(* IEC 61131-3 sources: Word/plc-course/13-sequential-control/labs/starter, 3 files *)

(* ---- 13-1-pedestrian-crossing.st ---- *)
(* Lab 13-1: Pedestrian crossing as a CASE state machine.
   Module 13 (Sequential control). STARTER - the declarations are done for you;
   write the logic where it says TODO, then run:
     python3 tools/plctest.py 13-sequential-control/labs/starter/13-1-pedestrian-crossing.st

   The enumeration, the state variables and the step timer are suggestions:
   the test only looks at the I/O and the settings, so you may organise the
   internals differently. *)

TYPE
  E_Crossing : (Startup, RedAmber, Green, Amber, AllRed, Walk, PedClear);
END_TYPE

PROGRAM PedCrossing
  VAR (* I/O *)
    PedPB    AT %IX0.0 : BOOL;  (* pedestrian request push-button, NO *)
    CarRed   AT %QX0.0 : BOOL;  (* vehicle signal, red *)
    CarAmber AT %QX0.1 : BOOL;  (* vehicle signal, amber *)
    CarGreen AT %QX0.2 : BOOL;  (* vehicle signal, green *)
    PedRed   AT %QX0.3 : BOOL;  (* pedestrian signal, red figure: do not cross *)
    PedGreen AT %QX0.4 : BOOL;  (* pedestrian signal, green figure: cross *)
    WaitLamp AT %QX0.5 : BOOL;  (* WAIT lamp on the push-button box *)
  END_VAR
  VAR (* settings *)
    StartupTime  : TIME := T#3s;   (* all red after power-up *)
    RedAmberTime : TIME := T#2s;   (* red + amber before green *)
    MinGreen     : TIME := T#10s;  (* minimum vehicle green *)
    AmberTime    : TIME := T#3s;   (* amber after green *)
    AllRedTime   : TIME := T#2s;   (* all red before the walk phase *)
    WalkTime     : TIME := T#6s;   (* steady green figure *)
    PedClearTime : TIME := T#4s;   (* flashing green figure *)
  END_VAR
  VAR (* internal - add your own helper variables here *)
    State      : E_Crossing := E_Crossing#Startup;
    PrevState  : E_Crossing := E_Crossing#Startup;
    FirstScan  : BOOL := TRUE;
    StepEntry  : BOOL;           (* TRUE on the first scan in a state *)
    StepTimer  : TON;            (* time spent in the current state *)
    Request    : BOOL;           (* latched pedestrian request *)
    FlashTimer : TON;            (* 500 ms flasher for the clearance phase *)
    FlashOn    : BOOL;
  END_VAR

  (* TODO: replace these placeholder lines with your logic.
     1. Step bookkeeping: StepEntry and StepTimer (reset on every change).
     2. CASE State OF ... with the transitions of each state.
     3. The request latch and the flasher.
     4. One assignment per output, derived from State. *)
  CarRed := TRUE;
  CarAmber := FALSE;
  CarGreen := FALSE;
  PedRed := TRUE;
  PedGreen := FALSE;
  WaitLamp := FALSE;
END_PROGRAM

CONFIGURATION Config0
  RESOURCE Res0 ON PLC
    TASK MainTask(INTERVAL := T#10ms, PRIORITY := 0);
    PROGRAM Inst0 WITH MainTask : PedCrossing;
  END_RESOURCE
END_CONFIGURATION

(* ---- 13-2-batch-tank.st ---- *)
(* Lab 13-2: Batch tank sequence with watchdogs, Hold/Resume and Abort.
   Module 13 (Sequential control). STARTER - the declarations are done for you;
   write the logic where it says TODO, then run:
     python3 tools/plctest.py 13-sequential-control/labs/starter/13-2-batch-tank.st

   The enumeration and the internal variables are suggestions: the test only
   looks at the I/O, TankTemp, the settings, FaultCode and BatchCount. *)

TYPE
  E_Batch : (Idle, Filling, Mixing, Heating, Draining, Complete, Held, Faulted);
END_TYPE

PROGRAM BatchTank
  VAR (* I/O *)
    StartPB      AT %IX0.0 : BOOL;  (* start a batch, NO *)
    HoldPB       AT %IX0.1 : BOOL;  (* hold the batch, NO *)
    ResumePB     AT %IX0.2 : BOOL;  (* resume a held batch, NO *)
    AbortPB      AT %IX0.3 : BOOL;  (* abort the batch, NO *)
    ResetPB      AT %IX0.4 : BOOL;  (* fault reset, NO *)
    LevelHighLS  AT %IX0.5 : BOOL;  (* high-level switch: TRUE when the tank is full *)
    LevelLowLS   AT %IX0.6 : BOOL;  (* low-level switch: TRUE while liquid covers it (and the heater) *)
    InletValve   AT %QX0.0 : BOOL;  (* fill valve *)
    Agitator     AT %QX0.1 : BOOL;  (* mixer motor *)
    Heater       AT %QX0.2 : BOOL;  (* immersion heater contactor *)
    OutletValve  AT %QX0.3 : BOOL;  (* drain valve *)
    RunLamp      AT %QX0.4 : BOOL;  (* batch running *)
    HeldLamp     AT %QX0.5 : BOOL;  (* batch held *)
    FaultLamp    AT %QX0.6 : BOOL;  (* sequence fault *)
    CompleteLamp AT %QX0.7 : BOOL;  (* batch complete *)
  END_VAR
  VAR (* process value, written by the analog-input layer (Module 14) *)
    TankTemp : REAL;                (* tank temperature, degC *)
  END_VAR
  VAR (* settings *)
    TempSP       : REAL := 60.0;    (* heat until TankTemp >= TempSP *)
    MixTime      : TIME := T#10s;   (* total mixing time *)
    FillTimeout  : TIME := T#30s;   (* watchdog: filling *)
    HeatTimeout  : TIME := T#60s;   (* watchdog: heating *)
    DrainTimeout : TIME := T#30s;   (* watchdog: draining *)
  END_VAR
  VAR (* status for the HMI *)
    FaultCode  : INT;               (* 0 none, 1 fill, 2 heat, 3 drain timeout *)
    BatchCount : INT;               (* completed batches *)
  END_VAR
  VAR (* internal - suggestions; add or change as you like *)
    State     : E_Batch := Idle;
    PrevState : E_Batch := Idle;
    HeldFrom  : E_Batch := Idle;  (* the step to resume *)
    FirstScan : BOOL := TRUE;
    StepEntry : BOOL;               (* TRUE on the first scan in a state *)
    StepTimer : TON;                (* time in the current state *)
    MixDone   : TIME;               (* mixing completed before a hold *)
    Running   : BOOL;               (* in one of the four process steps *)
    (* One instance per line: OpenPLC's compiler can crash on a list of
       FB instances in one declaration (see Appendix E). *)
    StartEdge : R_TRIG;
    HoldEdge : R_TRIG;
    ResumeEdge : R_TRIG;
    AbortEdge : R_TRIG;
    ResetEdge : R_TRIG;
    StartCmd, HoldCmd, ResumeCmd, AbortCmd, ResetCmd : BOOL;
  END_VAR

  (* TODO: replace these placeholder lines with your logic.
     1. Operator commands on the rising edge (R_TRIG).
     2. Step bookkeeping: StepEntry and StepTimer, reset on every change.
     3. Entry actions (BatchCount), before the transitions.
     4. Transitions: Abort first, then Hold, then CASE State OF ...
        with a watchdog in Filling, Heating and Draining.
     5. One assignment per output, derived from State, plus the heater and
        inlet interlocks. *)
  InletValve := FALSE;
  Agitator := FALSE;
  Heater := FALSE;
  OutletValve := FALSE;
  RunLamp := FALSE;
  HeldLamp := FALSE;
  FaultLamp := FALSE;
  CompleteLamp := FALSE;
END_PROGRAM

CONFIGURATION Config0
  RESOURCE Res0 ON PLC
    TASK MainTask(INTERVAL := T#10ms, PRIORITY := 0);
    PROGRAM Inst0 WITH MainTask : BatchTank;
  END_RESOURCE
END_CONFIGURATION

(* ---- 13-3-drill-sfc.st ---- *)
(* Lab 13-3: Drilling station in textual SFC, with action qualifiers.
   Module 13 (Sequential control). STARTER - the declarations are done for you;
   write the chart where it says TODO, then run:
     python3 tools/plctest.py 13-sequential-control/labs/starter/13-3-drill-sfc.st

   The program body is a Sequential Function Chart in the textual form of
   IEC 61131-3. Only the initial step is written so far. Add the steps,
   transitions and actions described in the lab, for example:

     STEP Clamp:
       ClampValve(S);
     END_STEP

     TRANSITION FROM Idle TO Clamp
       := StartPB AND PartPE AND DrillUpLS;
     END_TRANSITION

     ACTION CountHole:
       HoleCount := HoleCount + 1;
     END_ACTION

   Remember: a step name cannot be the same as a variable name, and two
   transitions leaving the same step must never be TRUE together. *)

PROGRAM DrillCycle
  VAR (* I/O *)
    StartPB     AT %IX0.0 : BOOL;  (* cycle start push-button, NO *)
    PartPE      AT %IX0.1 : BOOL;  (* part present in the fixture *)
    ClampedLS   AT %IX0.2 : BOOL;  (* clamp closed *)
    DrillUpLS   AT %IX0.3 : BOOL;  (* drill head at the top (home) *)
    DrillDownLS AT %IX0.4 : BOOL;  (* drill at full depth *)
    ResetPB     AT %IX0.5 : BOOL;  (* fault reset push-button, NO *)
    ClampValve  AT %QX0.0 : BOOL;  (* clamp solenoid valve: TRUE = clamp *)
    Spindle     AT %QX0.1 : BOOL;  (* spindle motor contactor *)
    FeedDown    AT %QX0.2 : BOOL;  (* feed valve, down *)
    FeedUp      AT %QX0.3 : BOOL;  (* feed valve, up (neither = hold position) *)
    BlowAir     AT %QX0.4 : BOOL;  (* chip blow-off air valve *)
    ReadyLamp   AT %QX0.5 : BOOL;  (* ready for a new part *)
    FaultLamp   AT %QX0.6 : BOOL;  (* feed fault *)
  END_VAR
  VAR (* settings and counters *)
    SpinUpTime  : TIME := T#500ms; (* spindle run-up before the feed starts *)
    DwellTime   : TIME := T#1s;    (* dwell at full depth *)
    BlowTime    : TIME := T#1s;    (* longest blow-off during the retract *)
    FeedTimeout : TIME := T#5s;    (* longest time allowed to reach depth *)
    HoleCount   : INT;             (* holes drilled to full depth *)
  END_VAR

  INITIAL_STEP Idle:
    ReadyLamp(N);
  END_STEP

  (* TODO: the rest of the chart: Clamp, Drill, Dwell, Retract, Unclamp,
     Unload, and the FeedFault branch, with their transitions and the
     action qualifiers N, S, R, D, L and P. *)
END_PROGRAM

CONFIGURATION Config0
  RESOURCE Res0 ON PLC
    TASK MainTask(INTERVAL := T#10ms, PRIORITY := 0);
    PROGRAM Inst0 WITH MainTask : DrillCycle;
  END_RESOURCE
END_CONFIGURATION
